FUNCTION_BLOCK process
VAR_INPUT
END_VAR
VAR_OUTPUT
END_VAR
VAR
END_VAR

END_FUNCTION_BLOCK

(* stored: Version 1.1.0.1, ProductVersion 3.1.4024.12
   POU process: Id {0b46f966-e3dd-410d-b569-329a8f71ea39}, SpecialFunc None *)
